// TIA Portal V15.1 export
// export: Created 2024-05-17T05:38:25.5609276Z, ExportSetting WithDefaults, DisplayName Totally Integrated Automation Portal, DisplayVersion V15.1 Update 5, DisplayName TIA Portal Openness, DisplayVersion V15.1 Update 5, DisplayName SINAMICS Startdrive Advanced, DisplayVersion V15.1, DisplayName G130, G150, S120, S150, SINAMICS MV, S210, DisplayVersion V15.1, DisplayName G110M, G120, G120C, G120D, G120P, DisplayVersion V15.1, DisplayName STEP 7 Professional, DisplayVersion V15.1 Update 5, DisplayName STEP 7 Safety, DisplayVersion V15.1, DisplayName WinCC Professional, DisplayVersion V15.1 Update 5, DisplayName SIMATIC Visualization Architect, DisplayVersion V15.1
FUNCTION "LAlarmDword" : Void   // FC2107, FBD
TITLE = LAlarmDword
{ S7_Optimized_Access := 'TRUE' }
AUTHOR : VCC
FAMILY : Anim
VERSION : 0.0.0.0
// =============================================================================The function shall provide/prepare all the necessary data for the alarmhandling systems. This function shall act as the serving point and collect all alarm statusses from its level. =============================================================================
// stored: AutoNumber false, IsIECCheckEnabled false, SetENOAutomatically False, UDAEnableTagReadback false
   VAR_INPUT
      I_Alarm00 : Bool;   // Alarm 00
      I_Alarm01 : Bool;   // Alarm 01
      I_Alarm02 : Bool;   // Alarm 02
      I_Alarm03 : Bool;   // Alarm 03
      I_Alarm04 : Bool;   // Alarm 04
      I_Alarm05 : Bool;   // Alarm 05
      I_Alarm06 : Bool;   // Alarm 06
      I_Alarm07 : Bool;   // Alarm 07
      I_Alarm08 : Bool;   // Alarm 08
      I_Alarm09 : Bool;   // Alarm 09
      I_Alarm10 : Bool;   // Alarm 10
      I_Alarm11 : Bool;   // Alarm 11
      I_Alarm12 : Bool;   // Alarm 12
      I_Alarm13 : Bool;   // Alarm 13
      I_Alarm14 : Bool;   // Alarm 14
      I_Alarm15 : Bool;   // Alarm 15
      I_Alarm16 : Bool;   // Alarm 16
      I_Alarm17 : Bool;   // Alarm 17
      I_Alarm18 : Bool;   // Alarm 18
      I_Alarm19 : Bool;   // Alarm 19
      I_Alarm20 : Bool;   // Alarm 20
      I_Alarm21 : Bool;   // Alarm 21
      I_Alarm22 : Bool;   // Alarm 22
      I_Alarm23 : Bool;   // Alarm 23
      I_Alarm24 : Bool;   // Alarm 24
      I_Alarm25 : Bool;   // Alarm 25
      I_Alarm26 : Bool;   // Alarm 26
      I_Alarm27 : Bool;   // Alarm 27
      I_Alarm28 : Bool;   // Alarm 28
      I_Alarm29 : Bool;   // Alarm 29
      I_Alarm30 : Bool;   // Alarm 30
      I_Alarm31 : Bool;   // Alarm 31
   END_VAR
   VAR_OUTPUT
      H_AlarmDWord : DWord;   // Alarn DWord for HMI
   END_VAR
BEGIN

REGION Network 1: **** 8 - Outputs ****
   // Alarm
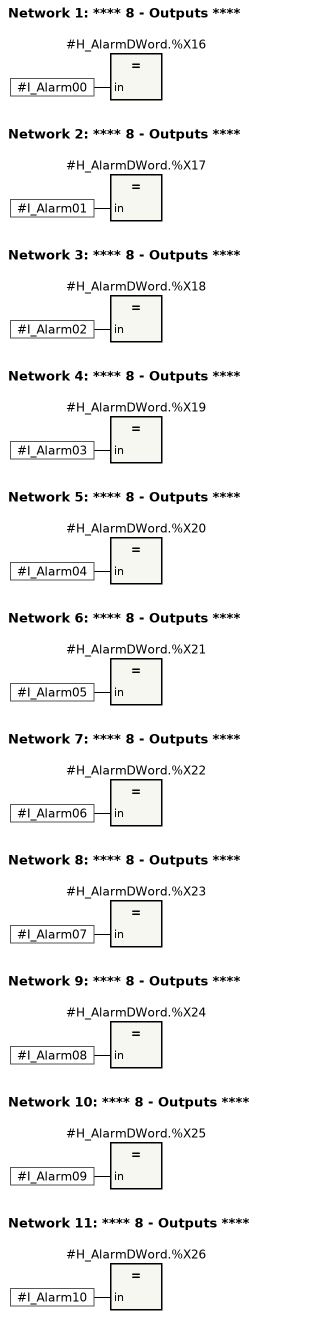
   #H_AlarmDWord.%X16 := #I_Alarm00;
END_REGION

REGION Network 2: **** 8 - Outputs ****
   // Alarm
   #H_AlarmDWord.%X17 := #I_Alarm01;
END_REGION

REGION Network 3: **** 8 - Outputs ****
   // Alarm
   #H_AlarmDWord.%X18 := #I_Alarm02;
END_REGION

REGION Network 4: **** 8 - Outputs ****
   // Alarm
   #H_AlarmDWord.%X19 := #I_Alarm03;
END_REGION

REGION Network 5: **** 8 - Outputs ****
   // Alarm
   #H_AlarmDWord.%X20 := #I_Alarm04;
END_REGION

REGION Network 6: **** 8 - Outputs ****
   // Alarm
   #H_AlarmDWord.%X21 := #I_Alarm05;
END_REGION

REGION Network 7: **** 8 - Outputs ****
   // Alarm
   #H_AlarmDWord.%X22 := #I_Alarm06;
END_REGION

REGION Network 8: **** 8 - Outputs ****
   // Alarm
   #H_AlarmDWord.%X23 := #I_Alarm07;
END_REGION

REGION Network 9: **** 8 - Outputs ****
   // Alarm
   #H_AlarmDWord.%X24 := #I_Alarm08;
END_REGION

REGION Network 10: **** 8 - Outputs ****
   // Alarm
   #H_AlarmDWord.%X25 := #I_Alarm09;
END_REGION

REGION Network 11: **** 8 - Outputs ****
   // Alarm
   #H_AlarmDWord.%X26 := #I_Alarm10;
END_REGION

REGION Network 12: **** 8 - Outputs ****
   // Alarm
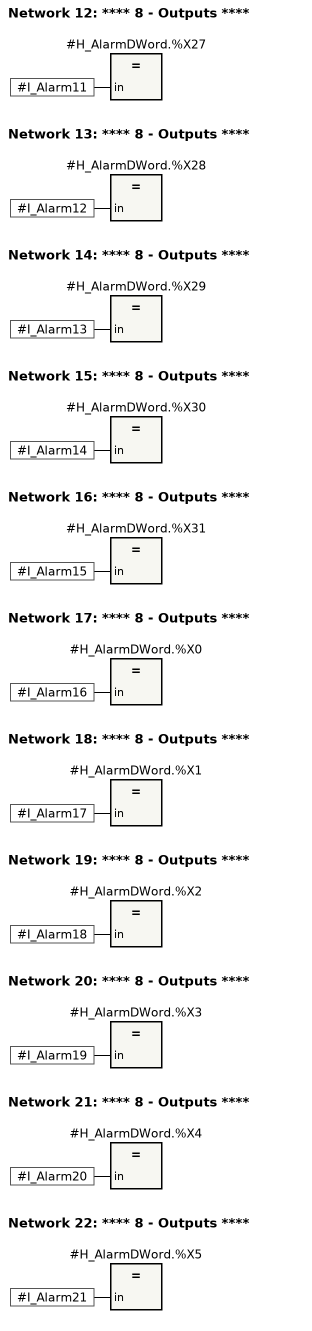
   #H_AlarmDWord.%X27 := #I_Alarm11;
END_REGION

REGION Network 13: **** 8 - Outputs ****
   // Alarm
   #H_AlarmDWord.%X28 := #I_Alarm12;
END_REGION

REGION Network 14: **** 8 - Outputs ****
   // Alarm
   #H_AlarmDWord.%X29 := #I_Alarm13;
END_REGION

REGION Network 15: **** 8 - Outputs ****
   // Alarm
   #H_AlarmDWord.%X30 := #I_Alarm14;
END_REGION

REGION Network 16: **** 8 - Outputs ****
   // Alarm
   #H_AlarmDWord.%X31 := #I_Alarm15;
END_REGION

REGION Network 17: **** 8 - Outputs ****
   // Alarm
   #H_AlarmDWord.%X0 := #I_Alarm16;
END_REGION

REGION Network 18: **** 8 - Outputs ****
   // Alarm
   #H_AlarmDWord.%X1 := #I_Alarm17;
END_REGION

REGION Network 19: **** 8 - Outputs ****
   // Alarm
   #H_AlarmDWord.%X2 := #I_Alarm18;
END_REGION

REGION Network 20: **** 8 - Outputs ****
   // Alarm
   #H_AlarmDWord.%X3 := #I_Alarm19;
END_REGION

REGION Network 21: **** 8 - Outputs ****
   // Alarm
   #H_AlarmDWord.%X4 := #I_Alarm20;
END_REGION

REGION Network 22: **** 8 - Outputs ****
   // Alarm
   #H_AlarmDWord.%X5 := #I_Alarm21;
END_REGION

REGION Network 23: **** 8 - Outputs ****
   // Alarm
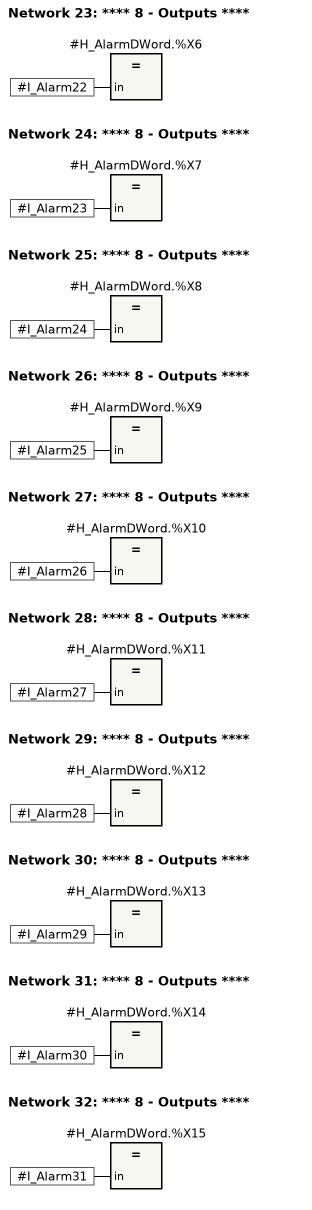
   #H_AlarmDWord.%X6 := #I_Alarm22;
END_REGION

REGION Network 24: **** 8 - Outputs ****
   // Alarm
   #H_AlarmDWord.%X7 := #I_Alarm23;
END_REGION

REGION Network 25: **** 8 - Outputs ****
   // Alarm
   #H_AlarmDWord.%X8 := #I_Alarm24;
END_REGION

REGION Network 26: **** 8 - Outputs ****
   // Alarm
   #H_AlarmDWord.%X9 := #I_Alarm25;
END_REGION

REGION Network 27: **** 8 - Outputs ****
   // Alarm
   #H_AlarmDWord.%X10 := #I_Alarm26;
END_REGION

REGION Network 28: **** 8 - Outputs ****
   // Alarm
   #H_AlarmDWord.%X11 := #I_Alarm27;
END_REGION

REGION Network 29: **** 8 - Outputs ****
   // Alarm
   #H_AlarmDWord.%X12 := #I_Alarm28;
END_REGION

REGION Network 30: **** 8 - Outputs ****
   // Alarm
   #H_AlarmDWord.%X13 := #I_Alarm29;
END_REGION

REGION Network 31: **** 8 - Outputs ****
   // Alarm
   #H_AlarmDWord.%X14 := #I_Alarm30;
END_REGION

REGION Network 32: **** 8 - Outputs ****
   // Alarm
   #H_AlarmDWord.%X15 := #I_Alarm31;
END_REGION
END_FUNCTION
